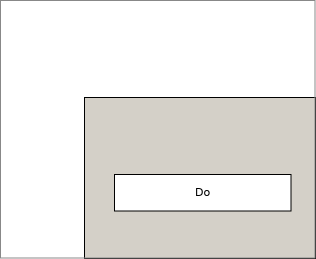
VISUALIZATION Test  // 316x259
    RoundedRectangle (84,97 232x162)
    RoundedRectangle (114,174 177x37), "Do"
        OnMouseClick: execute { Anlage.Gripper.DoSomething(); }
END_VISUALIZATION

(* stored: Version 1.1.0.1
   Visu Test: Id {61552118-6dd5-42b3-8f64-68d21c48a571} *)
